VISUALIZATION ManualMotionScreen  // 2x2
END_VISUALIZATION

(* stored: Version 1.1.0.1, ProductVersion 3.1.4024.13
   Visu ManualMotionScreen: Id {62b650f8-3ecf-4e21-a20c-fb31927f68c9} *)
